(* PLC project Unnamed, Unknown Unnamed 1 *)
(* stored: creationDateTime 2021-09-10T18:59:05, modificationDateTime 2021-09-29T07:23:11 *)

PROGRAM program0
  VAR
    p_red AT %QX100.0 : BOOL;
    p_green AT %QX100.1 : BOOL;
    v_red AT %QX100.2 : BOOL;
    v_yel AT %QX100.3 : BOOL;
    v_green AT %QX100.4 : BOOL;
    p_right AT %QX0.0 : BOOL;
    p_left AT %QX0.1 : BOOL;
    start AT %QX0.2 : BOOL;
  END_VAR
  VAR
    T2 : BOOL;
    T3 : BOOL;
    T4 : BOOL;
    T5 : BOOL;
    T6 : BOOL;
    TON0 : TON;
    TON1 : TON;
    TON2 : TON;
    TON3 : TON;
  END_VAR
  VAR
    C1 AT %MW1 : INT;
    C2 AT %MW2 : INT;
    C3 AT %MW3 : INT;
    C4 AT %MW4 : INT;
    C5 AT %MW5 : INT;
  END_VAR
  VAR
    TON4 : TON;
    TON5 : TON;
  END_VAR
  VAR  (* added by the conversion: wires and edge detectors of the diagram *)
    _TIME_TO_INT42_OUT : INT;
  END_VAR

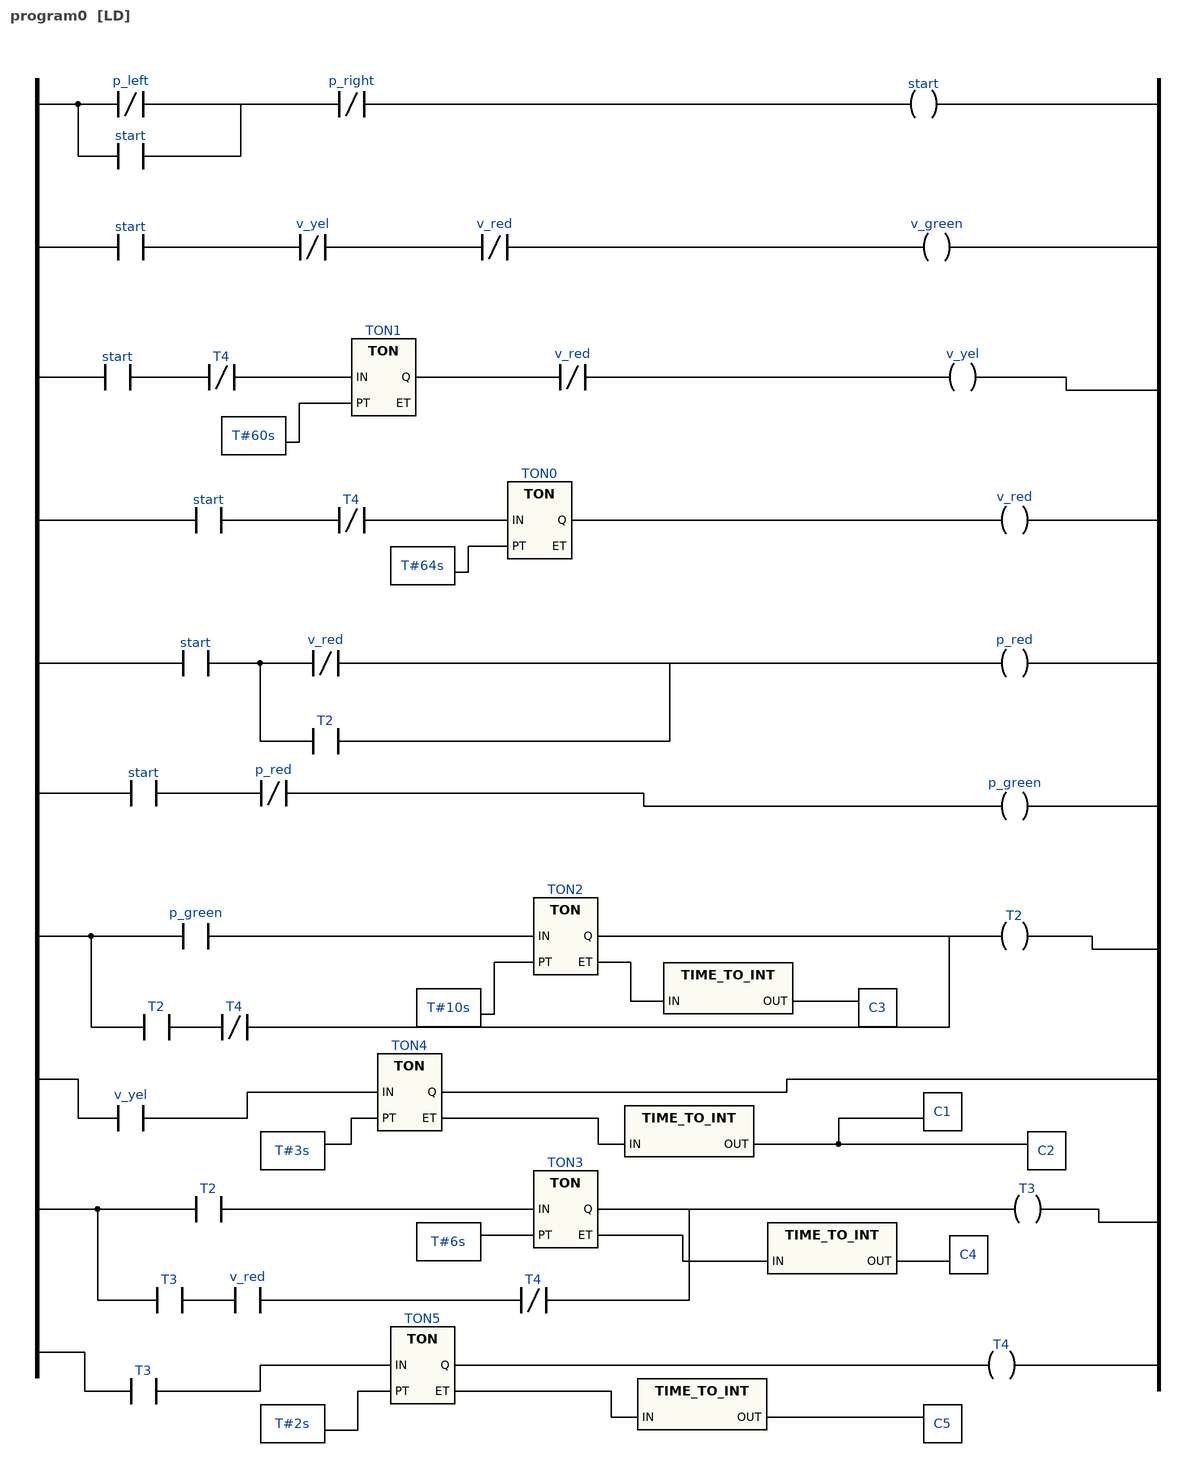
(* LD diagram, written out as Structured Text *)
start := (NOT p_left OR start) AND NOT p_right;
v_green := start AND NOT v_yel AND NOT v_red;
TON1(IN := start AND NOT T4, PT := T#60s);
v_yel := TON1.Q AND NOT v_red;
TON0(IN := start AND NOT T4, PT := T#64s);
v_red := TON0.Q;
p_red := start AND (NOT v_red OR T2);
p_green := start AND NOT p_red;
TON2(IN := p_green, PT := T#10s);
T2 := TON2.Q OR T2 AND NOT T4;
C3 := TIME_TO_INT(TON2.ET);
TON4(IN := v_yel, PT := T#3s);
_TIME_TO_INT42_OUT := TIME_TO_INT(TON4.ET);
C1 := _TIME_TO_INT42_OUT;
C2 := _TIME_TO_INT42_OUT;
TON3(IN := T2, PT := T#6s);
T3 := TON3.Q OR T3 AND v_red AND NOT T4;
C4 := TIME_TO_INT(TON3.ET);
TON5(IN := T3, PT := T#2s);
T4 := TON5.Q;
C5 := TIME_TO_INT(TON5.ET);
END_PROGRAM

CONFIGURATION Config0
  RESOURCE Res0 ON PLC
    TASK task0(INTERVAL := T#20ms, PRIORITY := 0);
    PROGRAM instance0 WITH task0 : program0;
  END_RESOURCE
END_CONFIGURATION
